FUNCTION_BLOCK WoodBunkEx_old
VAR_IN_OUT //controls
	execute : BOOL;
	stop : BOOL;
	
	manualStep : BOOL;
	manualSuction : BOOL;
END_VAR
VAR_IN_OUT //references to required hardware
	robotLeft, robotRight : RobotA21;
	toolStorageLeft, toolStorageRight : A21ToolStorage;
	
	stagingTableLeft, stagingTableRight : StagingTable;
	magazineLeft, magazineRight : SkidMagazine;
	
	strapper : StrapMachine;
	
	horizontalDriveLeft, horizontalDriveRight : AirPiston;
	verticalDriveLeft, verticalDriveRight : ClearLinkMC;
	pistonBottom : SimplePiston;
	
	suctionTop : ARRAY[*] OF SuctionPad; (*1..3*)
	suctionLeft : ARRAY[*] OF SuctionPad; (*1..4*)
	suctionRight : ARRAY[*] OF SuctionPad; (*1..4*)
	suctionBottom : ARRAY[*] OF SuctionPad; (*1..2*)
END_VAR
VAR_OUTPUT
	//ready : BOOL;
	done : BOOL;
	error : BOOL;
END_VAR
VAR //for testing, to be removed when deployoed
	latchLeft, latchRight : BOOL; //prevents SMC sliders from overshooting the inner limit sensor
	
	suctionEnableTop : BOOL;
	suctionEnableLeft : BOOL;
	suctionEnableRight : BOOL;
	suctionEnableBottom : BOOL;
END_VAR
VAR //Allen-Bradley-style AOIs encapsulate functionality and reduce the number of module variables
	templateLeft, templateRight : AOI_StagingTemplate;
	stageLeft, stageRight : AOI_StageWoodBunk; 
	loadLeft, loadRight : AOI_LoadWoodBunk;
	
	topSuctionDelay : TON;
	
	step : (IDLE, STAGING, LOAD_WB, PUSH, STRAP, RELEASE, COMPLETE := 1050);
	iPair : INT;
	
	loadStep : INT;
	stageStep : INT;
	iSlotLeft, iSlotRight : INT;
END_VAR
VAR //local types
	demoHeight : REAL := 600; //mm
	materialsArr : ARRAY[0..GVL.maxPairs] OF PositionMaterials := [
		(
			position := 0,
			top := 'WDS20', left := 'WDS20', right := 'WDS20', bottom := 'WDB20'
		),
		(
			position := 69,
			top := 'WDS20', left := 'WDS20', right := 'WDS20', bottom := 'WDB20'
		)];
	
	//stagingTemplateLeft, stagingTemplateRight AT %M* : StagingTable;
	//templateSlotsLeft, templateSlotsRight : ARRAY[1..10] OF STRING;
	//templateOccupancyLeft, templateOccupancyRight : ARRAY[1..10] OF BOOL;
	//stagingArrayLeft, stagingArrayRight : ARRAY[0..(GVL.maxPairs+1)*2] OF STRING;
	
	insertionLeft, insertionRight : Insertion;
	
	loadedMaterials : ARRAY[Surface.TOP..Surface.BOTTOM] OF STRING;
END_VAR
VAR CONSTANT
	sectionID : SectionEnum := SectionEnum.WOOD_BUNK;
END_VAR
VAR
	a,b,c,d : BOOL;
END_VAR

callLocalModules(); //initialize local modules

blocks(); //call local function blocks

IF robotRight.Done THEN
	robotRight.clearCommand();
END_IF

IF stop THEN
	stopSequence(); //stop everything
	RETURN;
END_IF

IF NOT insertionLeft.screw.HomeSet OR NOT insertionRight.screw.HomeSet THEN
	homingSequence(); //homing all motion devices and robots
	RETURN;
END_IF

a S= suctionTop[1].occupied AND suctionTop[2].occupied AND suctionTop[3].occupied;
b S= suctionLeft[1].occupied AND suctionLeft[2].occupied AND suctionLeft[3].occupied AND suctionLeft[4].occupied;
c S= suctionRight[1].occupied AND suctionRight[2].occupied AND suctionRight[3].occupied AND suctionRight[4].occupied;
d S= suctionBottom[1].occupied AND suctionBottom[2].occupied;

CASE step OF
	IDLE:
		IF execute THEN
			execute := FALSE;
			suctionEnableTop := suctionEnableLeft := suctionEnableRight := suctionEnableBottom := FALSE;
			step := STAGING;
		END_IF
		
		SetSuctions(suctionTop, suctionEnableTop);
		SetSuctions(suctionLeft, suctionEnableLeft);
		SetSuctions(suctionRight, suctionEnableRight);
		SetSuctions(suctionBottom, suctionEnableBottom);
		
	STAGING:
		IF NOT done THEN
			done := stage(error => error);
		END_IF
		
		IF
			(manualStep AND_THEN execute) OR
			(NOT manualStep AND_THEN done)
		THEN
			execute := FALSE;
			done := FALSE;
			step := LOAD_WB;
		END_IF
	
	LOAD_WB:
		IF NOT done THEN
			done := load(pairIndex := iPair, error => error);
		END_IF
		
		IF manualSuction THEN
			SetSuctions(suctionTop, suctionEnableTop);
			SetSuctions(suctionLeft, suctionEnableLeft);
			SetSuctions(suctionRight, suctionEnableRight);
			SetSuctions(suctionBottom, suctionEnableBottom);
		END_IF
		
		IF
			(manualStep AND_THEN execute) OR
			(NOT manualStep AND_THEN done)
		THEN
			done := FALSE;
			suctionEnableTop := suctionEnableLeft := suctionEnableRight := suctionEnableBottom := FALSE;
			execute := FALSE;
			
			step := PUSH;
		END_IF
		
	PUSH:
		IF
			(manualStep AND_THEN execute) OR
			(latchLeft AND latchRight AND pistonBottom.extended)
		THEN
			latchLeft := latchRight := FALSE;
			execute := FALSE;
			step := STRAP;
			RETURN;
		END_IF
		
		IF NOT validateSuctionQuality(checkTop:= TRUE, checkLeft:= TRUE, checkRight:= FALSE, checkBottom:= FALSE) THEN
			error := TRUE;
			RETURN;
		END_IF
		(*
		IF 
			insertionLeft.sliderPos <> demoHeight/2 //OR 
			//insertionRight.sliderPos <> demoHeight/2 //OR 
			//NOT insertionBottom.contact
		THEN
			insertionLeft.slideAbsolute(demoHeight/2);
			//insertionRight.slideAbsolute(demoHeight/2);
			RETURN;
		END_IF
		*)
		
		IF insertionLeft.screw.AtInnerLimit THEN
			latchLeft := TRUE;
		ELSIF NOT latchLeft THEN
			insertionLeft.press();
		END_IF
		
		IF insertionRight.screw.AtInnerLimit THEN
			latchRight := TRUE;
		ELSIF NOT latchRight THEN
			insertionRight.press();
		END_IF
		pistonBottom.extend();
		
	STRAP:
		topSuctionDelay(IN:= , PT:= T#1S, Q=> , ET=> );
		
		strapper.bEnable := TRUE;
		IF strapper.done THEN
			topSuctionDelay.IN := FALSE;
			step := RELEASE;
			RETURN;
		END_IF
		
		IF topSuctionDelay.Q THEN
			SetSuctions(suctionTop, FALSE);
			SetSuctions(suctionLeft, FALSE);
			SetSuctions(suctionRight, FALSE);
			SetSuctions(suctionBottom, FALSE);
		ELSIF strapper.atBundleLevel THEN
			topSuctionDelay.IN := TRUE;
		END_IF
		
		IF strapper.ready THEN
			strapper.strap();
		END_IF
		
		IF execute THEN
			topSuctionDelay.IN := FALSE;
			execute := FALSE;
			step := RELEASE;
		END_IF
		
	RELEASE: //release command		
		//insertionLeft.slideAbsolute(0);
		//insertionRight.slideAbsolute(0);
		
		insertionLeft.release();
		insertionRight.release();
		pistonBottom.retract();
		
		IF 
			(insertionLeft.screw.AtHome AND insertionRight.screw.AtHome AND pistonBottom.retracted) OR
			execute
		THEN
			execute := FALSE;
			step := COMPLETE;
		END_IF
	
	COMPLETE:
		//reset everything
		iPair := (iPair + 1) MOD GVL.maxPairs;
		step := IDLE;
		
		a := b := c := d := FALSE;
END_CASE

ACTION blocks:
templateLeft(
	execute:= , 
	materialsArr:= materialsArr, 
	table:= stagingTableLeft, 
	includeTop:= TRUE, 
	includeLeft:= TRUE, 
	includeRight:= FALSE, 
	includeBottom:= FALSE);

templateLeft(
	execute:= , 
	materialsArr:= materialsArr, 
	table:= stagingTableRight, 
	includeTop:= FALSE, 
	includeLeft:= FALSE, 
	includeRight:= TRUE, 
	includeBottom:= TRUE);
	
stageLeft(
	sectionID:= sectionID, 
	execute:= ,
	robot:= robotLeft, 
	table:= stagingTableLeft, 
	magazine:= magazineLeft, 
	slot:= iSlotLeft, 
	material:= templateLeft.getSlot(iSlotLeft), //stagingTemplateLeft.getSlot(iSlotRight), 
	done=> , 
	error=> );

stageRight(
	sectionID:= sectionID, 
	execute:= ,
	robot:= robotRight, 
	table:= stagingTableRight, 
	magazine:= magazineRight, 
	slot:= iSlotRight, 
	material:= stagingTemplateRight.getSlot(iSlotRight), 
	done=> , 
	error=> );

loadLeft(
	sectionID:= sectionID, 
	execute:= ,
	robot:= robotLeft, 
	table:= stagingTableLeft, 
	suctions:= suctionTop,
	loadedMaterials:= loadedMaterials,
	recoveryAoiStage:= stageLeft, 
	recoveryMagazine:= magazineLeft, 
	surfaceID:= , 
	material:= , 
	loadedMaterials=> , 
	done=> , 
	error=> );
	
loadRight(
	sectionID:= sectionID, 
	execute:= ,
	robot:= robotRight, 
	table:= stagingTableRight, 
	suctions:= suctionTop,
	loadedMaterials:= loadedMaterials,
	recoveryAoiStage:= stageRight, 
	recoveryMagazine:= magazineRight, 
	surfaceID:= , 
	material:= , 
	loadedMaterials=> , 
	done=> , 
	error=> );
END_ACTION

ACTION callLocalModules:
{warning disable C0371}
stagingTemplateLeft(slots := templateSlotsLeft, occupied := templateOccupancyLeft);
stagingTemplateRight(slots := templateSlotsRight, occupied := templateOccupancyRight);

insertionLeft(
	enable:= TRUE, 
	slider:= verticalDriveLeft, 
	screw:= horizontalDriveLeft, 
	contact=> , 
	softContact=> , 
	busy=> , 
	error=> , 
	home=> , 
	homingComplete=> , 
	sliderPos=> );
	
insertionRight(
	enable:= TRUE, 
	slider:= verticalDriveRight, 
	screw:= horizontalDriveRight,  
	contact=> , 
	softContact=> , 
	busy=> , 
	error=> , 
	home=> , 
	homingComplete=> , 
	sliderPos=> );
END_ACTION

METHOD createStagingArrayLeft : BOOL
VAR
	remainingMaterial : STRING;
	splitMaterial : STRING;
	
	i : INT;
END_VAR
FOR i:=0 TO (GVL.maxPairs+1)*2 BY 1 DO
	remainingMaterial := materialsArr[i].top;
	WHILE FIND(remainingMaterial, '_') > 0 DO
		splitCombinedMaterials(remainingMaterial, splitMaterial);
		IF splitMaterial <> '' THEN
			AddToStringArray(arr := stagingArrayLeft, newString := splitMaterial, numElements => , nextIndex => );
		END_IF
	END_WHILE
	
	IF remainingMaterial <> '' THEN
		AddToStringArray(arr := stagingArrayLeft, newString := remainingMaterial, numElements => , nextIndex => );
	END_IF
	
	
	remainingMaterial := materialsArr[i].left;
	WHILE FIND(remainingMaterial, '_') > 0 DO
		splitCombinedMaterials(remainingMaterial, splitMaterial);
		IF splitMaterial <> '' THEN
			AddToStringArray(arr := stagingArrayLeft, newString := splitMaterial, numElements => , nextIndex => );
		END_IF
	END_WHILE
	
	IF remainingMaterial <> '' THEN
		AddToStringArray(arr := stagingArrayLeft, newString := remainingMaterial, numElements => , nextIndex => );
	END_IF
END_FOR
END_METHOD

METHOD createStagingArrayRight : BOOL
VAR
	remainingMaterial : STRING;
	splitMaterial : STRING;
	
	i : INT;
END_VAR
FOR i:=0 TO (GVL.maxPairs+1)*2 BY 1 DO
	remainingMaterial := materialsArr[i].bottom;
	WHILE FIND(remainingMaterial, '_') > 0 DO
		splitCombinedMaterials(remainingMaterial, splitMaterial);
		IF splitMaterial <> '' THEN
			AddToStringArray(arr := stagingArrayRight, newString := splitMaterial, numElements => , nextIndex => );
		END_IF
	END_WHILE
	
	IF remainingMaterial <> '' THEN
		AddToStringArray(arr := stagingArrayRight, newString := remainingMaterial, numElements => , nextIndex => );
	END_IF
	
	
	
	remainingMaterial := materialsArr[i].right;
	WHILE FIND(remainingMaterial, '_') > 0 DO
		splitCombinedMaterials(remainingMaterial, splitMaterial);
		IF splitMaterial <> '' THEN
			AddToStringArray(arr := stagingArrayRight, newString := splitMaterial, numElements => , nextIndex => );
		END_IF
	END_WHILE
	
	IF remainingMaterial <> '' THEN
		AddToStringArray(arr := stagingArrayRight, newString := remainingMaterial, numElements => , nextIndex => );
	END_IF
END_FOR
END_METHOD

METHOD PROTECTED generateStagingTemplate : BOOL
VAR
	i : INT;
END_VAR
createStagingArrayLeft();
createStagingArrayRight();

(*
iterate through all pairs and autofill the template
replace succesfully autofilled materials with empty string

when staging needs to be performed a 2nd time, autofilling empty strings is always unsuccessful
*)
FOR i:=0 TO (GVL.maxPairs+1)*2 BY 1 DO
	IF stagingTemplateLeft.autofill(materialID := stagingArrayLeft[i]) THEN
		stagingArrayLeft[i] := '';
	END_IF
	
	IF stagingTemplateRight.autofill(materialID := stagingArrayRight[i]) THEN
		stagingArrayRight[i] := '';
	END_IF
END_FOR

generateStagingTemplate := TRUE;
END_METHOD

ACTION homingSequence:
insertionLeft.homingSequence();
insertionRight.homingSequence();
pistonBottom.retract();
END_ACTION

METHOD PROTECTED load : BOOL
VAR_INPUT
	pairIndex : INT;
END_VAR
VAR_OUTPUT
	error : BOOL;
END_VAR
VAR
	pair : REFERENCE TO PositionMaterials REF= materialsArr[pairIndex];
END_VAR
{warning disable C0371}

CASE loadStep OF
	0: //top and bottom
		IF loadLeft.done AND loadRight.done THEN
			loadLeft.reset();
			loadRight.reset();
			
			loadLeft.execute := loadRight.execute := FALSE;
			loadStep := 10;
			RETURN;
		END_IF
		
		loadLeft.suctions := suctionTop;
		loadLeft.material := pair.top;
		
		loadRight.suctions := suctionBottom;
		loadRight.material := pair.bottom;
		
		loadLeft.execute := loadRight.execute := TRUE;
		
	10: //sides
		IF loadLeft.done AND loadRight.done THEN
			loadLeft.reset();
			loadRight.reset();
			
			loadLeft.execute := loadRight.execute := FALSE;
			loadStep := COMPLETE;
			RETURN;
		END_IF
		
		loadLeft.suctions := suctionLeft;
		loadLeft.material := pair.left;
		
		loadRight.suctions := suctionRight;
		loadRight.material := pair.right;
		
		loadLeft.execute := loadRight.execute := TRUE;
		
	COMPLETE:				
		robotLeft.release(sectionID);
		robotRight.release(sectionID);
		
		loadLeft.execute := loadRight.execute := FALSE;
		
		loadStep := 0;
		load := TRUE;
END_CASE
	
error := loadLeft.error OR loadRight.error;
END_METHOD

METHOD splitCombinedMaterials : BOOL
VAR_IN_OUT
	materialID : STRING;
	splitMaterial : STRING;
END_VAR
VAR
	i : INT;
END_VAR
FindAndSplitChar(
	sSeparatorChar:= '_', 
	pSrcString:= ADR(materialID), 
	
	pLeftString:= ADR(splitMaterial), 
	nLeftSize:= SIZEOF(splitMaterial), 
	
	pRightString:= ADR(materialID), 
	nRightSize:= SIZEOF(materialID), 
	
	bSearchFromRight:= FALSE);
END_METHOD

METHOD stage : BOOL
VAR_OUTPUT
	error : BOOL;
END_VAR
{warning disable C0371}

CASE stageStep OF
	0: //generate staging template
		generateStagingTemplate();
		stageStep := 10;
		RETURN;
		
		IF templateLeft.done THEN
			templateLeft.execute := FALSE;
			
		END_IF
		
	10: //stage tables
		IF iSlotLeft > 10 AND iSlotRight > 10 THEN
			stageStep := COMPLETE;
			stageLeft.execute := stageRight.execute := FALSE;
			RETURN;
		END_IF
		
		stageLeft.execute := stageRight.execute := TRUE;
		
		//--------------------------------------------
		
		iSlotLeft := MAX(1, iSlotLeft); //if 0, sets to 1
		iSlotLeft := MIN(iSLotLeft, 10); //if 11, sets to 10 before reincrements back to 11
		
		IF stageLeft.done THEN
			iSlotLeft := iSlotLeft + 1;
			stageLeft.reset();
		END_IF
		
		//--------------------------------------------
		
		iSlotRight := MAX(1, iSlotRight);
		iSlotRight := MIN(iSlotRight, 10);
		
		IF stageRight.done THEN
			iSlotRight := iSlotRight + 1;
			stageRight.reset();
		END_IF
	
	COMPLETE:
		stageLeft.reset();
		stageRight.reset();
		
		robotLeft.release(sectionID);
		robotRight.release(sectionID);
		
		stageLeft.execute := stageRight.execute := FALSE;
		iSlotLeft := iSlotRight := 0;
		
		stage := TRUE;
END_CASE

error := stageLeft.error OR stageRight.error;
END_METHOD

ACTION stopSequence:
insertionLeft.stop();
insertionRight.stop();
pistonBottom.stop();

robotLeft.clearCommand();
robotRight.clearCommand();

//stop conveyors
END_ACTION

METHOD validateSuctionQuality : BOOL
VAR_INPUT
	checkTop : BOOL;
	checkLeft : BOOL;
	checkRight : BOOL;
	checkBottom : BOOL;
END_VAR
validateSuctionQuality := 
	(NOT checkTop OR_ELSE SuctionQuality(suctions:= suctionTop)) AND
	(NOT checkLeft OR_ELSE SuctionQuality(suctions:= suctionLeft)) AND
	(NOT checkRight OR_ELSE SuctionQuality(suctions:= suctionRight)) AND
	(NOT checkBottom OR_ELSE SuctionQuality(suctions:= suctionBottom));

(*
validateSuctionQuality := 
	(
		NOT checkTop OR_ELSE InsertionQuality(
			suctions:= suctionTop, 
			insertionMaterial:= loadedMaterials[Surface.TOP], 
			recipeMaterial:= materialsArr[iPair].top)
	) AND
	(
		NOT checkLeft OR_ELSE InsertionQuality(
			suctions:= suctionLeft, 
			insertionMaterial:= loadedMaterials[Surface.LEFT], 
			recipeMaterial:= materialsArr[iPair].left)
	) AND
	(
		NOT checkRight OR_ELSE InsertionQuality(
			suctions:= suctionRight, 
			insertionMaterial:= loadedMaterials[Surface.RIGHT], 
			recipeMaterial:= materialsArr[iPair].right)
	) AND
	(
		NOT checkBottom OR_ELSE InsertionQuality(
			suctions:= suctionBottom, 
			insertionMaterial:= loadedMaterials[Surface.BOTTOM], 
			recipeMaterial:= materialsArr[iPair].bottom)
	);
*)
END_METHOD

END_FUNCTION_BLOCK

(* stored: Version 1.1.0.1, ProductVersion 3.1.4024.11
   POU WoodBunkEx_old: Id {2088e8c4-0288-48d0-bf5f-a9e21e220f9a}, SpecialFunc None
   Folder Actions: Id {8905af30-d273-495a-8298-bf5d1c948e98}
   Folder Template: Id {09d5c311-4c3f-47ff-a4ee-978c10d79e0b}
   Action blocks: Id {f0b9988a-1f41-42ab-9dfe-0901aeb64aa0}
   Action callLocalModules: Id {9f6de33f-3696-42ba-98fb-1d7f5838bb74}
   Method createStagingArrayLeft: Id {e7b2b38f-28b7-4ca1-97db-f5642f9138ea}
   Method createStagingArrayRight: Id {a23fbf27-fc10-4125-87b3-bfb41c98b9d8}
   Method generateStagingTemplate: Id {f9c44c47-10b1-4c48-b55f-a72ead5d0dd8}
   Action homingSequence: Id {434a2267-66b1-4552-9d2d-9e49da7500b6}
   Method load: Id {8d72f845-77bd-4833-8bd3-efb9da6c3eb6}
   Method splitCombinedMaterials: Id {5100a1ce-9f09-44e8-a796-baee79f8eccf}
   Method stage: Id {369c79cb-d891-48d3-8b40-a140641ca5ca}
   Action stopSequence: Id {502b7e8e-3928-4ce8-afd1-e8d916fdb8d6}
   Method validateSuctionQuality: Id {db8770c6-aea3-4e2f-a689-e3c1905a8195} *)
